(*

short summary
=============

.. <legal notes>

legal notes
=================
| SPDX-FileCopyrightText: © 2023 ekvip automation GmbH <info@ekvip.de>
| SPDX-License-Identifier: Apache-2.0
| For details check: Apache-2.0_

.. _Apache-2.0: https://www.apache.org/licenses/LICENSE-2.0

.. </legal notes>

enumeration values
==================

*)

{warning 'header is generated please add your documentation'}
{attribute 'qualified_only'}
{attribute 'strict'}
{attribute 'to_string'}
TYPE FunctionType :
(
	EXACT 	:= 0,
	MAXIMUM := 1,
	MINIMUM	:= 2 
);
END_TYPE

(* stored: Version 1.1.0.1, ProductVersion 3.1.4024.12
   DUT FunctionType: Id {3e19cb2f-c3f8-4934-8aad-bca942a13fb2} *)
